// Return TRUE on any error value.
// Optionally carries the value over to nOut for further processing.
FUNCTION IsErr : BOOL
VAR_INPUT
    nIn : Result; // Result variable to check for an error
END_VAR
VAR_OUTPUT
    nOut : Result; // Carries the input value for further use
END_VAR

IsErr := nIn < 0;
nOut := nIn;

END_FUNCTION

(* stored: Version 1.1.0.1
   POU IsErr: Id {52bb3ec0-2300-4aef-8f80-2640742ad572}, SpecialFunc None *)
